(* CODESYS project CintasSoplado.project
   Title: CintasSoplado
   Version: 0.0.0.0
   Author: serbogr1

Project tree, tasks and I/O mapping:
  MyController : TM241CE40R, Schneider Electric, order no. TM241CE40R, version 4.0.6.18
    application Application
      task MAST (cyclic, interval 20 ms, priority 15, watchdog 100 ms x 1) calls ProcesoUno, ProcesoDos, Pulsadores
      global variables GVL
      program MyPOU [FBD]
      visualisation HMIW_Control
      image pool ImagePool
      program ProcesoDos [SFC]: E2_active, E8_active
      program ProcesoUno [SFC]: E8_active, E7_active, E9_active, E10_active, E11_active, E12_active
      program Pulsadores [LD]
    DI : Digital Inputs, Schneider Electric, version 4.0.6.18
        input  idwDI_IDW0 : DWORD  // IDW0
        input  ibDI_IB1 : BYTE  // IB1
    DQ : Digital Outputs, Schneider Electric, version 4.0.6.18
        output qwDQ_QW0 : WORD  // QW0
        output qbDQ_QB1 : BYTE  // QB1
    Counters : Counters, Schneider Electric, version 4.0.6.18
    Pulse_Generators : Pulse Generators, Schneider Electric, version 4.0.6.18
    Cartridge_1 : Cartridge, Schneider Electric, version 4.0.6.18
    Cartridge_2 : Cartridge, Schneider Electric, version 4.0.6.18
    IO_Bus : IO bus - TM3, Schneider Electric, version 4.0.6.18
    COM_Bus : COM bus, Schneider Electric, version 4.0.6.18
    Ethernet_1 : Ethernet Network, Schneider Electric, version 4.0.6.18
        settings: WebServer = TRUE; FTP Server = TRUE; SoMachine Protocol = TRUE; Modbus Server = TRUE; NetManage Protocol = TRUE; SNMP protocol = TRUE; Enable Routing = FALSE; WebVisu protocol = TRUE; DHCP Server Active = FALSE
    Serial_Line_1 : Serial line, Schneider Electric, version 4.0.6.18
      SoMachine_Network_Manager : SoMachine-Network Manager, Schneider Electric, version 4.0.0.2
    Serial_Line_2 : Serial line, Schneider Electric, version 4.0.6.18
      Modbus_Manager : Modbus Manager, Schneider Electric, version 4.0.0.2
  text list GlobalTextList
*)

// MyController/Application/GVL
VAR_GLOBAL
END_VAR

// MyController/Application/ProcesoUno
PROGRAM ProcesoUno
VAR
	bS_FC_Empujador_1          AT %IX0.0: BOOL; (*I1*)
	bS_IC_Empujador_1          AT %IX0.1: BOOL; (*I2*)
	bS_FC_Empujador_2          AT %IX0.2: BOOL; (*I3*)
	bS_IC_Empujador_2          AT %IX0.3: BOOL; (*I4*)
	bS_FT_Empujador_1          AT %IX0.4: BOOL; (*I5*)
	bS_FT_Fresadora            AT %IX0.5: BOOL; (*I6*)
	bS_FT_Carga                AT %IX0.6: BOOL; (*I7*)
	bS_FT_Taladro              AT %IX0.7: BOOL; (*I8*)
	bS_FT_Salida               AT %IX1.0: BOOL; (*I9*)
	
	bA_M_Empujador_1_Adelante  AT %QX0.4: BOOL; (*Q1*)
	bA_M_Empujador_1_Atras     AT %QX0.5: BOOL; (*Q2*)
	bA_M_Empujador_2_Adelante  AT %QX0.6: BOOL; (*Q3*)
	bA_M_Empujador_2_Atras     AT %QX0.7: BOOL; (*Q4*)
	bA_M_Cinta_Alimentacion    AT %QX1.0: BOOL; (*Q5*)
	bA_M_Cinta_Fresadora       AT %QX1.1: BOOL; (*Q6*)
	bA_M_Fresadora             AT %QX1.2: BOOL; (*Q7*)
	bA_M_Cinta_Taladro         AT %QX1.3: BOOL; (*Q8*)
	bA_M_Taladro               AT %QX1.4: BOOL; (*Q9*)
	bA_M_Cinta_Salida          AT %QX1.5: BOOL; (*Q10*)
	bA_Habilitar_Sistema       AT %QX1.6: BOOL; (*Q11*)
	
	bBotonEncendidoHMI         AT %IX1.1: BOOL; (*Boton Inicio HMI*)
	bBotonEmergenciaHMIW                : BOOL; (*Boton Inicio HMIW*)	
	bBotonInicioHMI            AT %IX1.2: BOOL; (*Boton Inicio HMI*)
	bBotonInicioHMIW                    : BOOL; (*Boton Inicio HMIW*)
    bBotonPiezaHMIW            AT %QX1.7: BOOL; (*Boton Poner Pieza*)
    bSiguientePieza            AT %QX0.3: BOOL; (*Activa cuando se puede poner la siguiente pieza*)	
	bFinSoplado                         : BOOL; (*Activa Cuando termina Soplado*)
	r_T_Fresado                         : INT:=1;
	r_T_Taladrado                       : INT:=1;

END_VAR

VAR_OUTPUT
	tEmpujador_1   : TIME:=T#1S;
	tFresado       : TIME:=T#1S;
	(*tTaladrado     : TIME:=T#1S;*)
	tEmpujador_2   : TIME:=T#2200MS;
END_VAR

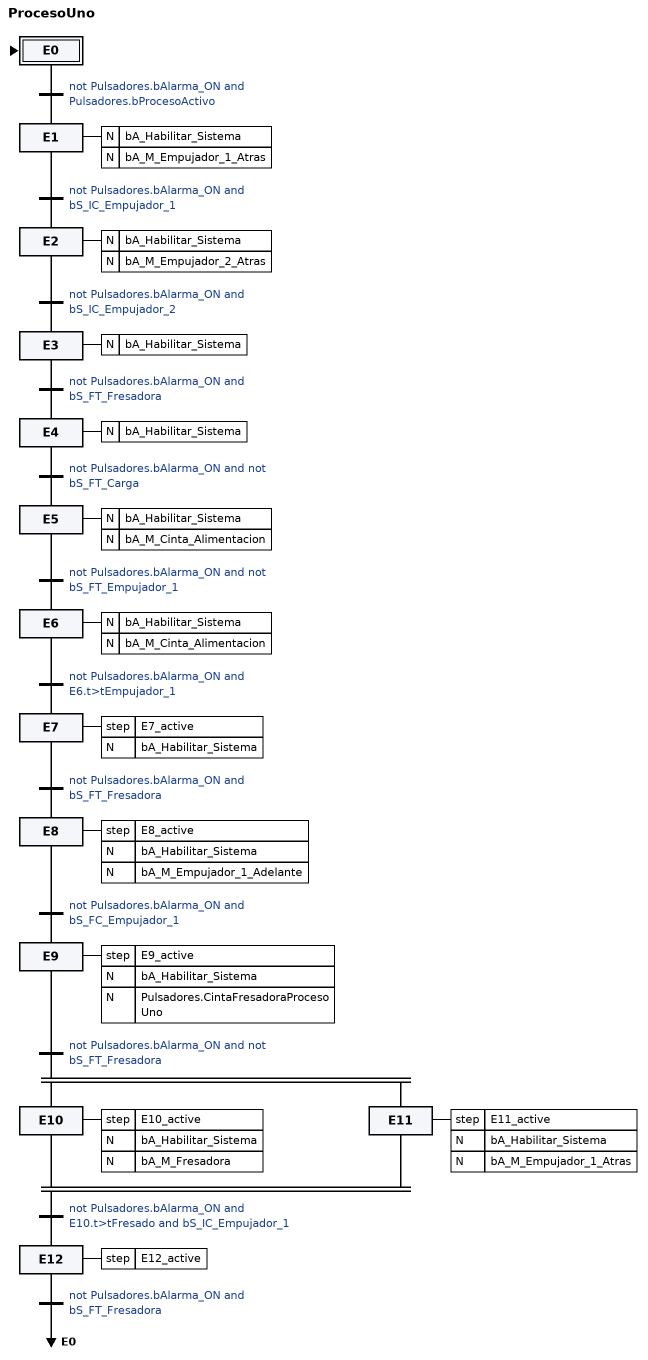
INITIAL_STEP E0:
END_STEP
TRANSITION FROM E0 TO E1
    := not Pulsadores.bAlarma_ON and Pulsadores.bProcesoActivo;
END_TRANSITION
STEP E1:
    bA_Habilitar_Sistema(N);
    bA_M_Empujador_1_Atras(N);
END_STEP
TRANSITION FROM E1 TO E2
    := not Pulsadores.bAlarma_ON and bS_IC_Empujador_1;
END_TRANSITION
STEP E2:
    bA_Habilitar_Sistema(N);
    bA_M_Empujador_2_Atras(N);
END_STEP
TRANSITION FROM E2 TO E3
    := not Pulsadores.bAlarma_ON and bS_IC_Empujador_2;
END_TRANSITION
STEP E3:
    bA_Habilitar_Sistema(N);
END_STEP
TRANSITION FROM E3 TO E4
    := not Pulsadores.bAlarma_ON and bS_FT_Fresadora;
END_TRANSITION
STEP E4:
    bA_Habilitar_Sistema(N);
END_STEP
TRANSITION FROM E4 TO E5
    := not Pulsadores.bAlarma_ON and not bS_FT_Carga;
END_TRANSITION
STEP E5:
    bA_Habilitar_Sistema(N);
    bA_M_Cinta_Alimentacion(N);
END_STEP
TRANSITION FROM E5 TO E6
    := not Pulsadores.bAlarma_ON and not bS_FT_Empujador_1;
END_TRANSITION
STEP E6:
    bA_Habilitar_Sistema(N);
    bA_M_Cinta_Alimentacion(N);
END_STEP
TRANSITION FROM E6 TO E7
    := not Pulsadores.bAlarma_ON and E6.t>tEmpujador_1;
END_TRANSITION
STEP E7:
    E7_active(N);  // step action
    bA_Habilitar_Sistema(N);
END_STEP
TRANSITION FROM E7 TO E8
    := not Pulsadores.bAlarma_ON and bS_FT_Fresadora;
END_TRANSITION
STEP E8:
    E8_active(N);  // step action
    bA_Habilitar_Sistema(N);
    bA_M_Empujador_1_Adelante(N);
END_STEP
TRANSITION FROM E8 TO E9
    := not Pulsadores.bAlarma_ON and bS_FC_Empujador_1;
END_TRANSITION
STEP E9:
    E9_active(N);  // step action
    bA_Habilitar_Sistema(N);
    Pulsadores.CintaFresadoraProcesoUno(N);
END_STEP
TRANSITION FROM E9 TO (E10, E11)
    := not Pulsadores.bAlarma_ON and not bS_FT_Fresadora;
END_TRANSITION
STEP E10:
    E10_active(N);  // step action
    bA_Habilitar_Sistema(N);
    bA_M_Fresadora(N);
END_STEP
STEP E11:
    E11_active(N);  // step action
    bA_Habilitar_Sistema(N);
    bA_M_Empujador_1_Atras(N);
END_STEP
TRANSITION FROM (E10, E11) TO E12
    := not Pulsadores.bAlarma_ON and E10.t>tFresado and bS_IC_Empujador_1;
END_TRANSITION
STEP E12:
    E12_active(N);  // step action
END_STEP
TRANSITION FROM E12 TO E0
    := not Pulsadores.bAlarma_ON and bS_FT_Fresadora;
END_TRANSITION

ACTION E8_active:
IF bS_FT_Carga THEN
	bSiguientePieza := TRUE;
ELSIF NOT bS_FT_Carga THEN
	bSiguientePieza := FALSE;
END_IF
END_ACTION

ACTION E7_active:
IF bS_FT_Carga THEN
	bSiguientePieza := TRUE;
ELSIF NOT bS_FT_Carga THEN
	bSiguientePieza := FALSE;
END_IF
END_ACTION

ACTION E9_active:
IF bS_FT_Carga THEN
	bSiguientePieza := TRUE;
ELSIF NOT bS_FT_Carga THEN
	bSiguientePieza := FALSE;
END_IF
END_ACTION

ACTION E10_active:
IF bS_FT_Carga THEN
	bSiguientePieza := TRUE;
ELSIF NOT bS_FT_Carga THEN
	bSiguientePieza := FALSE;
END_IF

    tFresado := INT_TO_TIME(r_T_Fresado*1000);
END_ACTION

ACTION E11_active:
IF bS_FT_Carga THEN
	bSiguientePieza := TRUE;
ELSIF NOT bS_FT_Carga THEN
	bSiguientePieza := FALSE;
END_IF
END_ACTION

ACTION E12_active:
IF bS_FT_Carga THEN
	bSiguientePieza := TRUE;
ELSIF NOT bS_FT_Carga THEN
	bSiguientePieza := FALSE;
END_IF
END_ACTION

END_PROGRAM

// MyController/Application/ProcesoDos
PROGRAM ProcesoDos
VAR
		tTaladrado         : TIME:=T#1S;
		rPiezasTerminadas : INT:=0;
END_VAR

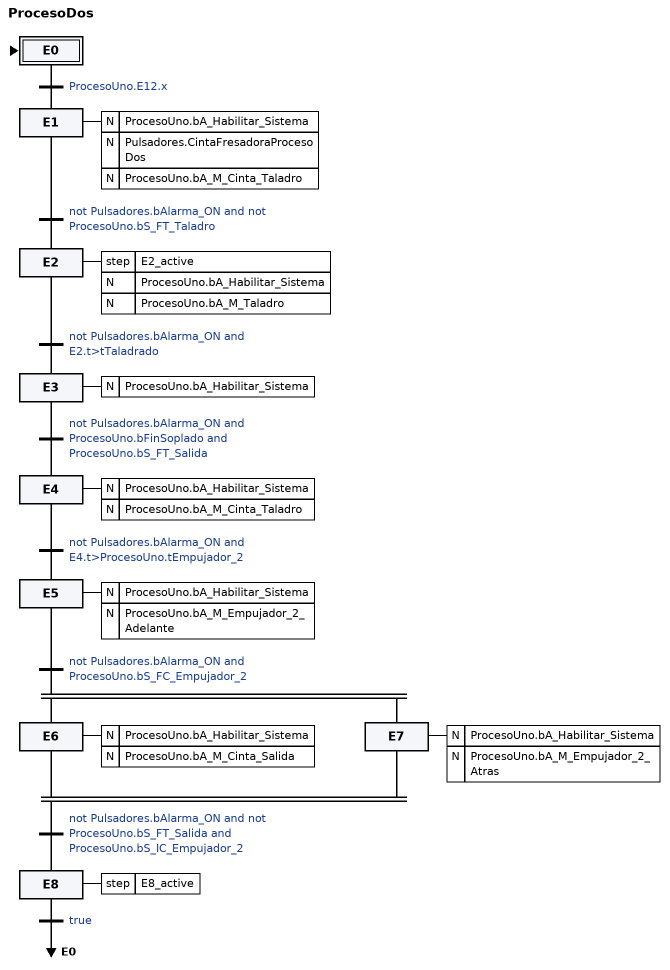
INITIAL_STEP E0:
END_STEP
TRANSITION FROM E0 TO E1
    := ProcesoUno.E12.x;
END_TRANSITION
STEP E1:
    ProcesoUno.bA_Habilitar_Sistema(N);
    Pulsadores.CintaFresadoraProcesoDos(N);
    ProcesoUno.bA_M_Cinta_Taladro(N);
END_STEP
TRANSITION FROM E1 TO E2
    := not Pulsadores.bAlarma_ON and not ProcesoUno.bS_FT_Taladro;
END_TRANSITION
STEP E2:
    E2_active(N);  // step action
    ProcesoUno.bA_Habilitar_Sistema(N);
    ProcesoUno.bA_M_Taladro(N);
END_STEP
TRANSITION FROM E2 TO E3
    := not Pulsadores.bAlarma_ON and E2.t>tTaladrado;
END_TRANSITION
STEP E3:
    ProcesoUno.bA_Habilitar_Sistema(N);
END_STEP
TRANSITION FROM E3 TO E4
    := not Pulsadores.bAlarma_ON and ProcesoUno.bFinSoplado and ProcesoUno.bS_FT_Salida;
END_TRANSITION
STEP E4:
    ProcesoUno.bA_Habilitar_Sistema(N);
    ProcesoUno.bA_M_Cinta_Taladro(N);
END_STEP
TRANSITION FROM E4 TO E5
    := not Pulsadores.bAlarma_ON and E4.t>ProcesoUno.tEmpujador_2;
END_TRANSITION
STEP E5:
    ProcesoUno.bA_Habilitar_Sistema(N);
    ProcesoUno.bA_M_Empujador_2_Adelante(N);
END_STEP
TRANSITION FROM E5 TO (E6, E7)
    := not Pulsadores.bAlarma_ON and ProcesoUno.bS_FC_Empujador_2;
END_TRANSITION
STEP E6:
    ProcesoUno.bA_Habilitar_Sistema(N);
    ProcesoUno.bA_M_Cinta_Salida(N);
END_STEP
STEP E7:
    ProcesoUno.bA_Habilitar_Sistema(N);
    ProcesoUno.bA_M_Empujador_2_Atras(N);
END_STEP
TRANSITION FROM (E6, E7) TO E8
    := not Pulsadores.bAlarma_ON and not ProcesoUno.bS_FT_Salida and ProcesoUno.bS_IC_Empujador_2;
END_TRANSITION
STEP E8:
    E8_active(N);  // step action
END_STEP
TRANSITION FROM E8 TO E0
    := true;
END_TRANSITION

ACTION E2_active:
  
tTaladrado := INT_TO_TIME(ProcesoUno.r_T_Taladrado*1000);
END_ACTION

ACTION E8_active:
IF NOT ProcesoUno.bS_FT_Salida THEN
	rPiezasTerminadas := rPiezasTerminadas + 1;
END_IF
END_ACTION

END_PROGRAM

// MyController/Application/Pulsadores
PROGRAM Pulsadores
VAR
	bAlarma_ON                          : BOOL; (*Activa cuando se pulsa alarma*)
	bProcesoActivo                      : BOOL;	(*Activa cuando se pulsa inicio*)	
	CintaFresadoraProcesoUno: BOOL;
	CintaFresadoraProcesoDos: BOOL;
	
	rLongTime: INT;
END_VAR

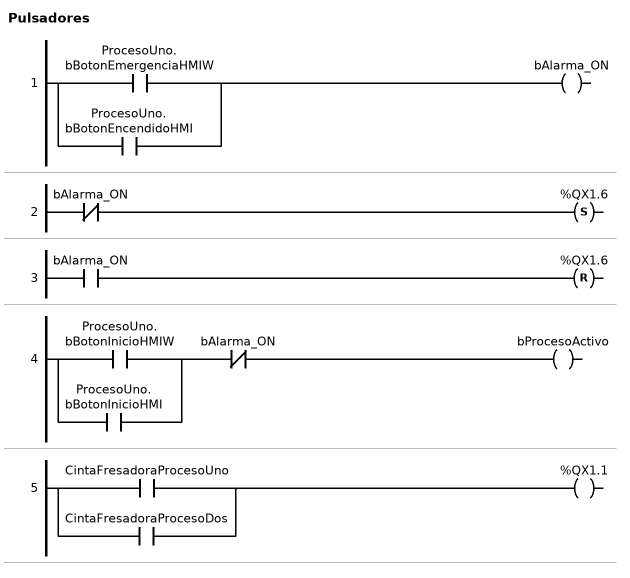
// NETWORK 1
bAlarma_ON := ProcesoUno.bBotonEmergenciaHMIW OR ProcesoUno.bBotonEncendidoHMI;

// NETWORK 2
%QX1.6 S= NOT bAlarma_ON;

// NETWORK 3
%QX1.6 R= bAlarma_ON;

// NETWORK 4
bProcesoActivo := (ProcesoUno.bBotonInicioHMIW OR ProcesoUno.bBotonInicioHMI) AND NOT bAlarma_ON;

// NETWORK 5
%QX1.1 := CintaFresadoraProcesoUno OR CintaFresadoraProcesoDos;

END_PROGRAM

// MyController/Application/MyPOU
PROGRAM MyPOU
VAR
END_VAR

// NETWORK 1

END_PROGRAM

// MyController/Application/HMIW_Control
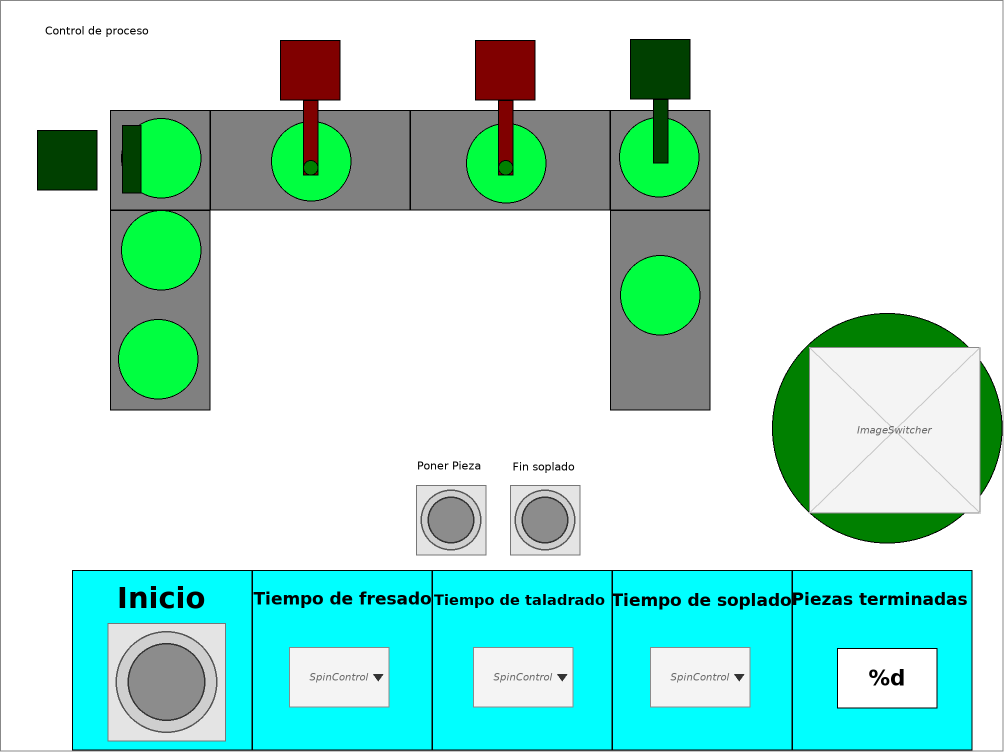
VISUALIZATION HMIW_Control  // 1004x752
    Ellipse (772,313 230x230), colour toggle: ProcesoUno.bBotonEmergenciaHMIW
    Label (22,16 150x30), "Control de proceso"
    Label (409,451 80x30), "Poner Pieza"
    PushSwitch (416,485 70x70), variable: ProcesoUno.bBotonPiezaHMIW, behaviour: TAP, style: Switch-PushSwitch-Gray
    PushSwitch (510,485 70x70), variable: ProcesoUno.bFinSoplado, behaviour: TAP, style: Switch-PushSwitch-Gray
    Label (504,452 79x30), "Fin soplado"
    Rectangle (72,570 180x180)
    Label (78,576 167x44), "Inicio"
    ImageSwitcher (809,347 171x166), variable: ProcesoUno.bBotonEmergenciaHMIW, background image: ImagePool.BotonEmergencia, image: ImagePool.BotonEmergencia, behaviour: TOGGLE
    Rectangle (252,570 180x180)
    SpinControl (289,647 100x60), variable: ProcesoUno.r_T_Fresado
    Rectangle (432,570 180x180)
    SpinControl (473,647 100x60), variable: ProcesoUno.r_T_Taladrado
    Rectangle (612,570 180x180)
    Label (609,585 185x30), "Tiempo de soplado"
    SpinControl (650,647 100x60)
    PushSwitchLed (103,623 127x118), variable: ProcesoUno.bBotonInicioHMIW, behaviour: TOGGLE, style: Switch-PushSwitchLed-Gray
    Label (256,574 173x49), "Tiempo de fresado"
    Label (423,569 193x62), "Tiempo de taladrado"
    Rectangle (110,210 100x200)
    Rectangle (110,110 100x100)
    Rectangle (210,110 200x100)
    Rectangle (410,110 200x100)
    Rectangle (610,110 100x100)
    Rectangle (610,210 100x200)
    Ellipse (118,319 80x80), invisible if: ProcesoUno.bS_FT_Carga
    Rectangle (792,570 180x180)
    Label (787,584 185x30), "Piezas terminadas"
    RoundedRectangle (837,648 100x60), "%d", text variable: ProcesoDos.rPiezasTerminadas
    RoundedRectangle (280,40 60x60)
    RoundedRectangle (475,40 60x60)
    Ellipse (121,210 80x80), invisible if: ProcesoUno.bS_FT_Empujador_1
    Ellipse (271,121 80x80), invisible if: ProcesoUno.bS_FT_Fresadora
    Rectangle (303,100 15x75)
    Ellipse (303,160 15x15), colour toggle: ProcesoUno.bA_M_Fresadora
    Ellipse (466,123 80x80), invisible if: ProcesoUno.bS_FT_Taladro
    Rectangle (498,100 15x75)
    Ellipse (498,160 15x15), colour toggle: ProcesoUno.bA_M_Taladro
    Ellipse (620,255 80x80), invisible if: ProcesoUno.bS_FT_Salida
    RoundedRectangle (630,39 60x60), colour toggle: ProcesoUno.bA_M_Empujador_2_Adelante
    Ellipse (619,117 80x80), invisible if: ProcesoUno.bS_IC_Empujador_2
    Rectangle (653,99 15x64), invisible if: not ProcesoUno.bA_M_Empujador_2_Adelante
    RoundedRectangle (37,130 60x60), colour toggle: ProcesoUno.bA_M_Empujador_1_Adelante
    Ellipse (121,118 80x80), invisible if: ProcesoUno.bS_IC_Empujador_1
    Rectangle (98,150 68x19), angle 90, invisible if: not ProcesoUno.bA_M_Empujador_1_Adelante
END_VISUALIZATION
